FUNCTION fc_RAD : real
VAR_INPUT
	DEG : REAL;
END_VAR
VAR
END_VAR

fc_RAD := fc_MODR(0.0174532925199433 * DEG, 6.28318530717958647692528676655900576);

END_FUNCTION

(* stored: Version 1.1.0.1, ProductVersion 3.1.4024.11
   POU fc_RAD: Id {cf0b0e06-347b-49c3-9074-948dee27f84b}, SpecialFunc None *)
